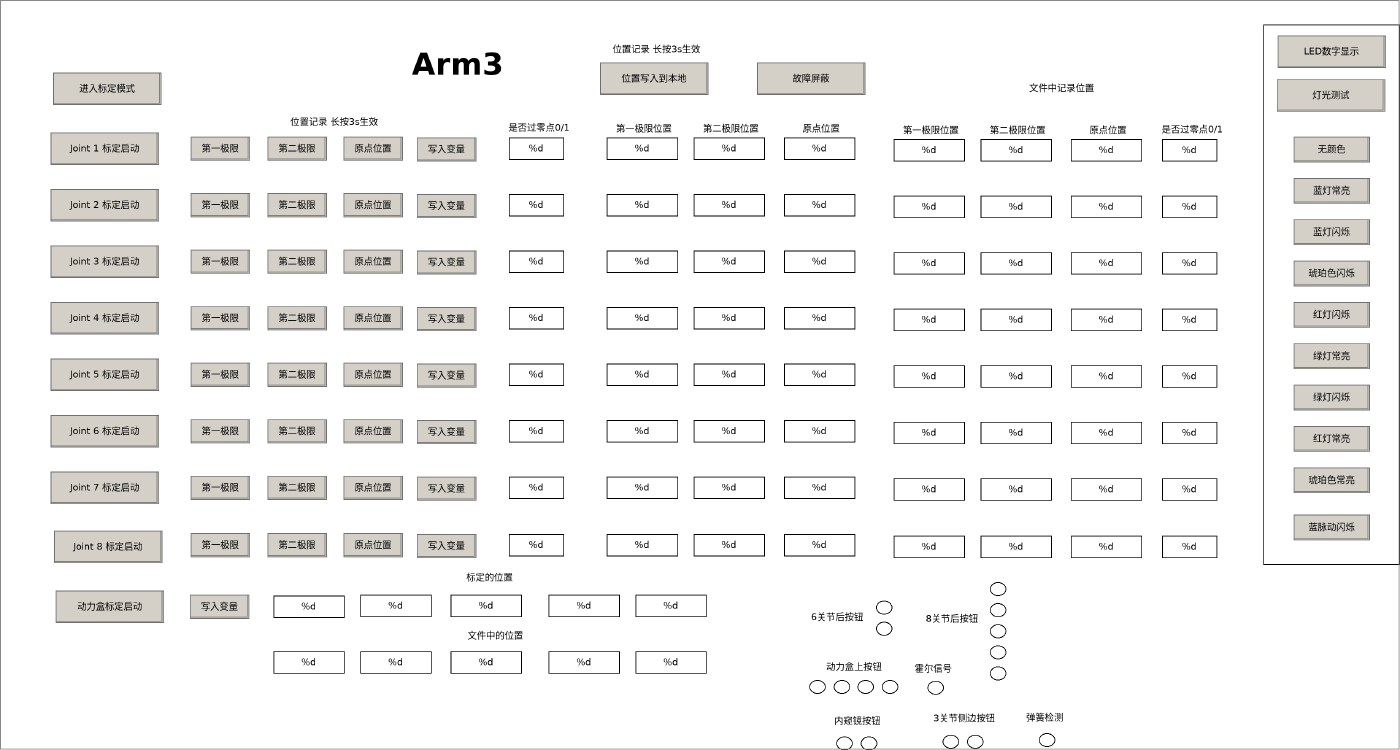
VISUALIZATION arm3Cail  // 1659x889
    Button (63,86 128x38), "进入标定模式", colour toggle: GVL_armCali.g_armEnterCaliMode[3]
        toggle GVL_armCali.g_armEnterCaliMode[3]
    Button (60,157 128x38), "Joint 1 标定启动", colour toggle: GVL_armCali.g_jointIntoCaliState[3][1]
        toggle GVL_armCali.g_jointIntoCaliState[3][1]
    Label (444,50 197x52), "Arm3"
    Button (60,224 128x38), "Joint 2 标定启动", colour toggle: GVL_armCali.g_jointIntoCaliState[3][2]
        toggle GVL_armCali.g_jointIntoCaliState[3][2]
    Button (226,162 70x28), "第一极限", colour toggle: GVL_armCali.g_linkEncFristCaliTrigger[3][1]
        tap GVL_armCali.g_linkEncFristPosCali[3][1]
    Button (317,162 70x28), "第二极限", colour toggle: GVL_armCali.g_linkEncSecondCaliTrigger[3][1]
        tap GVL_armCali.g_linkEncSecondPosCali[3][1]
    Rectangle (603,163 65x26), "%d", text variable: GVL_armCali.g_linkZeroCrossOrNot[3][1]
    Label (598,140 82x23), "是否过零点0/1"
    Rectangle (719,163 84x26), "%d", text variable: GVL_armCali.g_linkLimitFristPos[3][1]
    Label (722,141 82x23), "第一极限位置"
    Rectangle (822,163 84x26), "%d", text variable: GVL_armCali.g_linkLimitSecondPos[3][1]
    Label (825,141 82x23), "第二极限位置"
    Label (321,133 150x23), "位置记录 长按3s生效"
    Rectangle (929,163 84x26), "%d", text variable: GVL_armCali.g_linkHomePos[3][1]
    Label (932,141 82x23), "原点位置"
    Button (407,162 70x28), "原点位置", colour toggle: GVL_armCali.g_linkEncHomePosCaliTrigger[3][1]
        tap GVL_armCali.g_linkEncHomePosCali[3][1]
    Button (711,74 128x38), "位置写入到本地", colour toggle: GVL_armCali.g_caliDataWriteTrigger[3]
        tap GVL_armCali.g_caliDataWrite[3]
    Label (703,47 150x23), "位置记录 长按3s生效"
    Button (226,229 70x28), "第一极限", colour toggle: GVL_armCali.g_linkEncFristCaliTrigger[3][2]
        tap GVL_armCali.g_linkEncFristPosCali[3][2]
    Button (317,229 70x28), "第二极限", colour toggle: GVL_armCali.g_linkEncSecondCaliTrigger[3][2]
        tap GVL_armCali.g_linkEncSecondPosCali[3][2]
    Rectangle (603,230 65x26), "%d", text variable: GVL_armCali.g_linkZeroCrossOrNot[3][2]
    Rectangle (719,230 84x26), "%d", text variable: GVL_armCali.g_linkLimitFristPos[3][2]
    Rectangle (822,230 84x26), "%d", text variable: GVL_armCali.g_linkLimitSecondPos[3][2]
    Rectangle (929,230 84x26), "%d", text variable: GVL_armCali.g_linkHomePos[3][2]
    Button (407,229 70x28), "原点位置", colour toggle: GVL_armCali.g_linkEncHomePosCaliTrigger[3][2]
        tap GVL_armCali.g_linkEncHomePosCali[3][2]
    Button (60,291 128x38), "Joint 3 标定启动", colour toggle: GVL_armCali.g_jointIntoCaliState[3][3]
        toggle GVL_armCali.g_jointIntoCaliState[3][3]
    Button (226,296 70x28), "第一极限", colour toggle: GVL_armCali.g_linkEncFristCaliTrigger[3][3]
        tap GVL_armCali.g_linkEncFristPosCali[3][3]
    Button (317,296 70x28), "第二极限", colour toggle: GVL_armCali.g_linkEncSecondCaliTrigger[3][3]
        tap GVL_armCali.g_linkEncSecondPosCali[3][3]
    Rectangle (603,297 65x26), "%d", text variable: GVL_armCali.g_linkZeroCrossOrNot[3][3]
    Rectangle (719,297 84x26), "%d", text variable: GVL_armCali.g_linkLimitFristPos[3][3]
    Rectangle (822,297 84x26), "%d", text variable: GVL_armCali.g_linkLimitSecondPos[3][3]
    Rectangle (929,297 84x26), "%d", text variable: GVL_armCali.g_linkHomePos[3][3]
    Button (407,296 70x28), "原点位置", colour toggle: GVL_armCali.g_linkEncHomePosCaliTrigger[3][3]
        tap GVL_armCali.g_linkEncHomePosCali[3][3]
    Button (60,358 128x38), "Joint 4 标定启动", colour toggle: GVL_armCali.g_jointIntoCaliState[3][4]
        toggle GVL_armCali.g_jointIntoCaliState[3][4]
    Button (226,363 70x28), "第一极限", colour toggle: GVL_armCali.g_linkEncFristCaliTrigger[3][4]
        tap GVL_armCali.g_linkEncFristPosCali[3][4]
    Button (317,363 70x28), "第二极限", colour toggle: GVL_armCali.g_linkEncSecondCaliTrigger[3][4]
        tap GVL_armCali.g_linkEncSecondPosCali[3][4]
    Rectangle (603,364 65x26), "%d", text variable: GVL_armCali.g_linkZeroCrossOrNot[3][4]
    Rectangle (719,364 84x26), "%d", text variable: GVL_armCali.g_linkLimitFristPos[3][4]
    Rectangle (822,364 84x26), "%d", text variable: GVL_armCali.g_linkLimitSecondPos[3][4]
    Rectangle (929,364 84x26), "%d", text variable: GVL_armCali.g_linkHomePos[3][4]
    Button (407,363 70x28), "原点位置", colour toggle: GVL_armCali.g_linkEncHomePosCaliTrigger[3][4]
        tap GVL_armCali.g_linkEncHomePosCali[3][4]
    Button (60,425 128x38), "Joint 5 标定启动", colour toggle: GVL_armCali.g_jointIntoCaliState[3][5]
        toggle GVL_armCali.g_jointIntoCaliState[3][5]
    Button (226,430 70x28), "第一极限", colour toggle: GVL_armCali.g_linkEncFristCaliTrigger[3][5]
        tap GVL_armCali.g_linkEncFristPosCali[3][5]
    Button (317,430 70x28), "第二极限", colour toggle: GVL_armCali.g_linkEncSecondCaliTrigger[3][5]
        tap GVL_armCali.g_linkEncSecondPosCali[3][5]
    Rectangle (603,431 65x26), "%d", text variable: GVL_armCali.g_linkZeroCrossOrNot[3][5]
    Rectangle (719,431 84x26), "%d", text variable: GVL_armCali.g_linkLimitFristPos[3][5]
    Rectangle (822,431 84x26), "%d", text variable: GVL_armCali.g_linkLimitSecondPos[3][5]
    Rectangle (929,431 84x26), "%d", text variable: GVL_armCali.g_linkHomePos[3][5]
    Button (407,430 70x28), "原点位置", colour toggle: GVL_armCali.g_linkEncHomePosCaliTrigger[3][5]
        tap GVL_armCali.g_linkEncHomePosCali[3][5]
    Button (60,492 128x38), "Joint 6 标定启动", colour toggle: GVL_armCali.g_jointIntoCaliState[3][6]
        toggle GVL_armCali.g_jointIntoCaliState[3][6]
    Button (226,497 70x28), "第一极限", colour toggle: GVL_armCali.g_linkEncFristCaliTrigger[3][6]
        tap GVL_armCali.g_linkEncFristPosCali[3][6]
    Button (317,497 70x28), "第二极限", colour toggle: GVL_armCali.g_linkEncSecondCaliTrigger[3][6]
        tap GVL_armCali.g_linkEncSecondPosCali[3][6]
    Rectangle (603,498 65x26), "%d", text variable: GVL_armCali.g_linkZeroCrossOrNot[3][6]
    Rectangle (719,498 84x26), "%d", text variable: GVL_armCali.g_linkLimitFristPos[3][6]
    Rectangle (822,498 84x26), "%d", text variable: GVL_armCali.g_linkLimitSecondPos[3][6]
    Rectangle (929,498 84x26), "%d", text variable: GVL_armCali.g_linkHomePos[3][6]
    Button (407,497 70x28), "原点位置", colour toggle: GVL_armCali.g_linkEncHomePosCaliTrigger[3][6]
        tap GVL_armCali.g_linkEncHomePosCali[3][6]
    Button (60,559 128x38), "Joint 7 标定启动", colour toggle: GVL_armCali.g_jointIntoCaliState[3][7]
        toggle GVL_armCali.g_jointIntoCaliState[3][7]
    Button (226,564 70x28), "第一极限", colour toggle: GVL_armCali.g_linkEncFristCaliTrigger[3][7]
        tap GVL_armCali.g_linkEncFristPosCali[3][7]
    Button (317,564 70x28), "第二极限", colour toggle: GVL_armCali.g_linkEncSecondCaliTrigger[3][7]
        tap GVL_armCali.g_linkEncSecondPosCali[3][7]
    Rectangle (603,565 65x26), "%d", text variable: GVL_armCali.g_linkZeroCrossOrNot[3][7]
    Rectangle (719,565 84x26), "%d", text variable: GVL_armCali.g_linkLimitFristPos[3][7]
    Rectangle (822,565 84x26), "%d", text variable: GVL_armCali.g_linkLimitSecondPos[3][7]
    Rectangle (929,565 84x26), "%d", text variable: GVL_armCali.g_linkHomePos[3][7]
    Button (407,564 70x28), "原点位置", colour toggle: GVL_armCali.g_linkEncHomePosCaliTrigger[3][7]
        tap GVL_armCali.g_linkEncHomePosCali[3][7]
    Button (64,629 128x38), "Joint 8 标定启动", colour toggle: GVL_armCali.g_jointIntoCaliState[3][8]
        toggle GVL_armCali.g_jointIntoCaliState[3][8]
    Button (226,632 70x28), "第一极限", colour toggle: GVL_armCali.g_linkEncFristCaliTrigger[3][8]
        tap GVL_armCali.g_linkEncFristPosCali[3][8]
    Button (317,632 70x28), "第二极限", colour toggle: GVL_armCali.g_linkEncSecondCaliTrigger[3][8]
        tap GVL_armCali.g_linkEncSecondPosCali[3][8]
    Rectangle (603,633 65x26), "%d", text variable: GVL_armCali.g_linkZeroCrossOrNot[3][8]
    Rectangle (719,633 84x26), "%d", text variable: GVL_armCali.g_linkLimitFristPos[3][8]
    Rectangle (822,633 84x26), "%d", text variable: GVL_armCali.g_linkLimitSecondPos[3][8]
    Rectangle (929,633 84x26), "%d", text variable: GVL_armCali.g_linkHomePos[3][8]
    Button (407,632 70x28), "原点位置", colour toggle: GVL_armCali.g_linkEncHomePosCaliTrigger[3][8]
        tap GVL_armCali.g_linkEncHomePosCali[3][8]
    Rectangle (1059,165 84x26), "%d", text variable: GVL_SetupJointEncoderCaliData.g_minLinkEncoder[3,1]
    Label (1062,143 82x23), "第一极限位置"
    Rectangle (1162,165 84x26), "%d", text variable: GVL_SetupJointEncoderCaliData.g_maxLinkEncoder[3,1]
    Label (1165,143 82x23), "第二极限位置"
    Rectangle (1269,165 84x26), "%d", text variable: GVL_SetupJointEncoderCaliData.g_caliLinkEncoder[3,1]
    Label (1272,143 82x23), "原点位置"
    Rectangle (1059,232 84x26), "%d", text variable: GVL_SetupJointEncoderCaliData.g_minLinkEncoder[3,2]
    Rectangle (1162,232 84x26), "%d", text variable: GVL_SetupJointEncoderCaliData.g_maxLinkEncoder[3,2]
    Rectangle (1269,232 84x26), "%d", text variable: GVL_SetupJointEncoderCaliData.g_caliLinkEncoder[3,2]
    Rectangle (1059,299 84x26), "%d", text variable: GVL_SetupJointEncoderCaliData.g_minLinkEncoder[3,3]
    Rectangle (1162,299 84x26), "%d", text variable: GVL_SetupJointEncoderCaliData.g_maxLinkEncoder[3,3]
    Rectangle (1269,299 84x26), "%d", text variable: GVL_SetupJointEncoderCaliData.g_caliLinkEncoder[3,3]
    Rectangle (1059,366 84x26), "%d", text variable: GVL_SetupJointEncoderCaliData.g_minLinkEncoder[3,4]
    Rectangle (1162,366 84x26), "%d", text variable: GVL_SetupJointEncoderCaliData.g_maxLinkEncoder[3,4]
    Rectangle (1269,366 84x26), "%d", text variable: GVL_SetupJointEncoderCaliData.g_caliLinkEncoder[3,4]
    Rectangle (1059,433 84x26), "%d", text variable: GVL_SetupJointEncoderCaliData.g_minLinkEncoder[3,5]
    Rectangle (1162,433 84x26), "%d", text variable: GVL_SetupJointEncoderCaliData.g_maxLinkEncoder[3,5]
    Rectangle (1269,433 84x26), "%d", text variable: GVL_SetupJointEncoderCaliData.g_caliLinkEncoder[3,5]
    Rectangle (1059,500 84x26), "%d", text variable: GVL_SlaveJointEncoderCaliData.g_minLinkEncoder[3,1]
    Rectangle (1162,500 84x26), "%d", text variable: GVL_SlaveJointEncoderCaliData.g_maxLinkEncoder[3,1]
    Rectangle (1269,500 84x26), "%d", text variable: GVL_SlaveJointEncoderCaliData.g_caliLinkEncoder[3,1]
    Rectangle (1059,567 84x26), "%d", text variable: GVL_SlaveJointEncoderCaliData.g_minLinkEncoder[3,2]
    Rectangle (1162,567 84x26), "%d", text variable: GVL_SlaveJointEncoderCaliData.g_maxLinkEncoder[3,2]
    Rectangle (1269,567 84x26), "%d", text variable: GVL_SlaveJointEncoderCaliData.g_caliLinkEncoder[3,2]
    Rectangle (1059,635 84x26), "%d", text variable: GVL_SlaveJointEncoderCaliData.g_minLinkEncoder[3,3]
    Rectangle (1162,635 84x26), "%d", text variable: GVL_SlaveJointEncoderCaliData.g_maxLinkEncoder[3,3]
    Rectangle (1269,635 84x26), "%d", text variable: GVL_SlaveJointEncoderCaliData.g_caliLinkEncoder[3,3]
    Label (1183,93 150x23), "文件中记录位置"
    Rectangle (1377,165 65x26), "%d", text variable: GVL_SetupJointEncoderCaliData.g_linkEncZeroCross[3,1]
    Label (1372,142 82x23), "是否过零点0/1"
    Rectangle (1377,232 65x26), "%d", text variable: GVL_SetupJointEncoderCaliData.g_linkEncZeroCross[3,2]
    Rectangle (1377,299 65x26), "%d", text variable: GVL_SetupJointEncoderCaliData.g_linkEncZeroCross[3,3]
    Rectangle (1377,366 65x26), "%d", text variable: GVL_SetupJointEncoderCaliData.g_linkEncZeroCross[3,4]
    Rectangle (1377,433 65x26), "%d", text variable: GVL_SetupJointEncoderCaliData.g_linkEncZeroCross[3,5]
    Rectangle (1377,500 65x26), "%d", text variable: GVL_SlaveJointEncoderCaliData.g_linkEncZeroCross[3,1]
    Rectangle (1377,567 65x26), "%d", text variable: GVL_SlaveJointEncoderCaliData.g_linkEncZeroCross[3,2]
    Rectangle (1377,635 65x26), "%d", text variable: GVL_SlaveJointEncoderCaliData.g_linkEncZeroCross[3,3]
    Button (494,163 70x28), "写入变量", colour toggle: GVL_armCali.g_linkPosWriteCaliDataTrigger[3][1]
        tap GVL_armCali.g_linkPosWriteCaliData[3][1]
    Button (494,230 70x28), "写入变量", colour toggle: GVL_armCali.g_linkPosWriteCaliDataTrigger[3][2]
        tap GVL_armCali.g_linkPosWriteCaliData[3][2]
    Button (494,297 70x28), "写入变量", colour toggle: GVL_armCali.g_linkPosWriteCaliDataTrigger[3][3]
        tap GVL_armCali.g_linkPosWriteCaliData[3][3]
    Button (494,364 70x28), "写入变量", colour toggle: GVL_armCali.g_linkPosWriteCaliDataTrigger[3][4]
        tap GVL_armCali.g_linkPosWriteCaliData[3][4]
    Button (494,431 70x28), "写入变量", colour toggle: GVL_armCali.g_linkPosWriteCaliDataTrigger[3][5]
        tap GVL_armCali.g_linkPosWriteCaliData[3][5]
    Button (494,498 70x28), "写入变量", colour toggle: GVL_armCali.g_linkPosWriteCaliDataTrigger[3][6]
        tap GVL_armCali.g_linkPosWriteCaliData[3][6]
    Button (494,565 70x28), "写入变量", colour toggle: GVL_armCali.g_linkPosWriteCaliDataTrigger[3][7]
        tap GVL_armCali.g_linkPosWriteCaliData[3][7]
    Button (494,633 70x28), "写入变量", colour toggle: GVL_armCali.g_linkPosWriteCaliDataTrigger[3][8]
        tap GVL_armCali.g_linkPosWriteCaliData[3][8]
    Button (66,700 128x38), "动力盒标定启动", colour toggle: GVL_armCali.g_powerBoxCali[3]
        toggle GVL_armCali.g_powerBoxCali[3]
    Button (225,705 70x28), "写入变量", colour toggle: GVL_armCali.g_powerBoxPosWriteTrigger[3]
        tap GVL_armCali.g_powerBoxPosWrite[3]
    Rectangle (324,706 84x26), "%d", text variable: GVL_armCali.g_powerBoxLinkHomePos[3][1]
    Rectangle (427,705 84x26), "%d", text variable: GVL_armCali.g_powerBoxLinkHomePos[3][2]
    Rectangle (534,705 84x26), "%d", text variable: GVL_armCali.g_powerBoxLinkHomePos[3][3]
    Rectangle (650,705 84x26), "%d", text variable: GVL_armCali.g_powerBoxLinkHomePos[3][4]
    Rectangle (753,705 84x26), "%d", text variable: GVL_armCali.g_powerBoxLinkHomePos[3][5]
    Rectangle (324,772 84x26), "%d", text variable: GVL_SlaveJointEncoderCaliData.g_caliLinkEncoder[3,4]
    Rectangle (427,772 84x26), "%d", text variable: GVL_SlaveJointEncoderCaliData.g_caliLinkEncoder[3,5]
    Rectangle (534,772 84x26), "%d", text variable: GVL_SlaveJointEncoderCaliData.g_caliLinkEncoder[3,6]
    Rectangle (650,772 84x26), "%d", text variable: GVL_SlaveJointEncoderCaliData.g_caliLinkEncoder[3,7]
    Rectangle (753,772 84x26), "%d", text variable: GVL_SlaveJointEncoderCaliData.g_caliLinkEncoder[3,8]
    Label (512,742 150x23), "文件中的位置"
    Label (505,673 150x23), "标定的位置"
    Label (952,720 80x23), "6关节后按钮"
    Ellipse (1038,737 19x16), colour toggle: GVL_IO.g_joint6IO[3][2]
    Ellipse (1038,712 19x16), colour toggle: GVL_IO.g_joint6IO[3][1]
    Label (1088,722 80x23), "8关节后按钮"
    Ellipse (1173,715 19x16), colour toggle: GVL_IO.g_joint8IO[3][2]
    Ellipse (1173,690 19x16), colour toggle: GVL_IO.g_joint8IO[3][1]
    Ellipse (1173,765 19x16), colour toggle: GVL_IO.g_joint8IO[3][4]
    Ellipse (1173,740 19x16), colour toggle: GVL_IO.g_joint8IO[3][3]
    Label (972,779 80x23), "动力盒上按钮"
    Ellipse (959,806 19x16), colour toggle: GVL_IO.g_jointPowerBoxIO[3][1]
    Ellipse (988,806 19x16), colour toggle: GVL_IO.g_jointPowerBoxIO[3][2]
    Ellipse (1016,806 19x16), colour toggle: GVL_IO.g_jointPowerBoxIO[3][3]
    Ellipse (1045,806 19x16), colour toggle: GVL_IO.g_jointPowerBoxIO[3][4]
    Label (976,843 80x23), "内窥镜按钮"
    Ellipse (991,873 19x16), colour toggle: GVL_IO.g_endoscopeSingle[3][1]
    Ellipse (1020,873 19x16), colour toggle: GVL_IO.g_endoscopeSingle[3][2]
    Ellipse (1173,790 19x16), colour toggle: GVL_IO.g_joint8IO[3][5]
    Ellipse (1099,807 19x16), colour toggle: GVL_IO.g_jointPowerBoxIO[3][5]
    Label (1066,781 80x23), "霍尔信号"
    Rectangle (1497,29 162x640)
    Button (1533,162 90x30), "无颜色", colour toggle: GVL_IO.g_armLight_PowerOff[3]
        toggle GVL_IO.g_armLight_PowerOff[3]
    Button (1533,211 90x30), "蓝灯常亮", colour toggle: GVL_IO.g_armLight_BlueOn[3]
        toggle GVL_IO.g_armLight_BlueOn[3]
    Button (1533,260 90x30), "蓝灯闪烁", colour toggle: GVL_IO.g_armLight_BlueBlink[3]
        toggle GVL_IO.g_armLight_BlueBlink[3]
    Button (1533,309 90x30), "琥珀色闪烁", colour toggle: GVL_IO.g_armLight_AmberBlink[3]
        toggle GVL_IO.g_armLight_AmberBlink[3]
    Button (1533,358 90x30), "红灯闪烁", colour toggle: GVL_IO.g_armLight_RedBlink[3]
        toggle GVL_IO.g_armLight_RedBlink[3]
    Button (1533,407 90x30), "绿灯常亮", colour toggle: GVL_IO.g_armLight_GreenOn[3]
        toggle GVL_IO.g_armLight_GreenOn[3]
    Button (1533,456 90x30), "绿灯闪烁", colour toggle: GVL_IO.g_armLight_GreenBlink[3]
        toggle GVL_IO.g_armLight_GreenBlink[3]
    Button (1513,94 128x38), "灯光测试", colour toggle: GVL_IO.g_lightTest[3]
        toggle GVL_IO.g_lightTest[3]
    Button (1533,505 90x30), "红灯常亮", colour toggle: GVL_IO.g_armLight_redOn[3]
        toggle GVL_IO.g_armLight_redOn[3]
    Button (1533,554 90x30), "琥珀色常亮", colour toggle: GVL_IO.g_armLight_AmberOn[3]
        toggle GVL_IO.g_armLight_AmberOn[3]
    Button (1533,610 90x30), "蓝脉动闪烁", colour toggle: GVL_IO.g_armLight_BluePulse[3]
        toggle GVL_IO.g_armLight_BluePulse[3]
    Button (1514,42 128x38), "LED数字显示", colour toggle: GVL_IO.g_LEDValueDisplay[3]
        toggle GVL_IO.g_LEDValueDisplay[3]
    Label (1085,840 115x23), "3关节侧边按钮"
    Ellipse (1117,871 19x16), colour toggle: GVL_IO.g_asepticMegnetCheck[3][1]
    Ellipse (1146,871 19x16), colour toggle: GVL_IO.g_asepticMegnetCheck[3][2]
    Ellipse (1231,869 19x16)
    Label (1198,839 80x23), "弹簧检测"
    Button (897,74 128x38), "故障屏蔽", colour toggle: g_specialSignal.m_faultMask[3]
        toggle g_specialSignal.m_faultMask[3]
END_VISUALIZATION

(* stored: Version 1.1.0.1, ProductVersion 3.1.4024.11
   Visu arm3Cail: Id {065dbd63-4520-48dc-9ccc-64d7cf97ac3e} *)
